// TIA Portal V20 export
// export: Created 2025-12-01T14:57:00.3125225Z, ExportSetting None, DisplayName Totally Integrated Automation Portal, DisplayVersion V20 Update 3, DisplayName TIA Portal Openness, DisplayVersion V20 Update 3, DisplayName TIA Portal Version Control Interface, DisplayVersion V20 Update 3, DisplayName STEP 7 Professional, DisplayVersion V20 Update 3, DisplayName STEP 7 Safety, DisplayVersion V20 Update 2, DisplayName WinCC Basic/Comfort/Advanced, DisplayVersion V20 Update 3, DisplayName WinCC Professional, DisplayVersion V20 Update 3, DisplayName WinCC Unified, DisplayVersion V20 Update 3
FUNCTION "FC450_TL_TR_E1_S2_Pres" : Void   // FC450, LAD
{ S7_Optimized_Access := 'FALSE' }
AUTHOR : TLigero
NAME : 20160512
VERSION : 4.0
// stored: AutoNumber false, SetENOAutomatically false
   VAR_INPUT
      Mesa : UInt;
      En_Tension : Bool;
      PhsMx : Bool;
      Termico_E1 : Bool;
      Termico_S2 : Bool;
      PosTR_E1 : Bool;
      PosTR_S2 : Bool;
      Avance_E1 : Bool;
      Avance_S2 : Bool;
      AVTF_MAnt_Mx : Bool;   // Aviso de transferencia de la mesa anterior
      PTF_Mx_MSig : Bool;   // Permiso de transferencia de la mesa siguiente
      NXT_Avance : Bool;   // Avance de la mesa siguiente
      V_CNT_pHsMx : UDInt;
      V_CNT_ApHsMx : UDInt;
      V_Paro : UDInt;
      V_TOut_Tx_Mx : UDInt;
      V_TOut_transfer : UDInt;
   END_VAR
   VAR_OUTPUT
      PTF_MAnt_Mx : Bool;   // carga ok a la mesa anterior
      AVTF_Mx_MSig : Bool;   // Aviso de transferencia a la mesa siguiente
      NXT_Descarga_Act : Bool;   // descarga activa a la mesa siguiente
   END_VAR
   VAR_TEMP
      Mem_CNT_Tmp_Paro_Tx : Bool;
      Mem_CNT_Pres_entrada : Bool;
      Mem_CNT_Aus_salida : Bool;
      tout_atasco : Bool;
      tout_transfer : Bool;
      TEMP_MA_TR_Pos_E1 : Bool;
      TEMP_MA_TR_Pos_S2 : Bool;
      ok_tension : Bool;
   END_VAR
   VAR_TEMP   // added for the SCL form of the ladder/FBD networks
      _w1 : Bool;
   END_VAR
BEGIN

REGION Network 1: Marca General Error
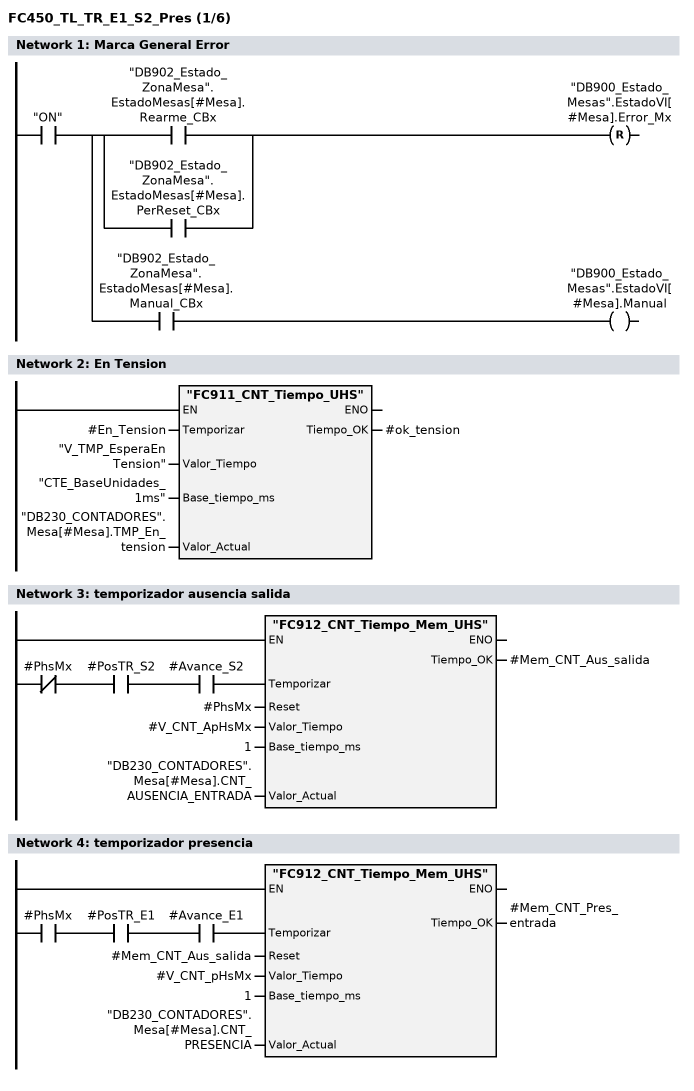
   RUNG wire#powerrail
      Contact( "ON" )
      wire#w1
      Contact( "DB902_Estado_ZonaMesa".EstadoMesas[#Mesa].Rearme_CBx )
      wire#w2
      R_Coil( "DB900_Estado_Mesas".EstadoVI[#Mesa].Error_Mx )
   END_RUNG
   RUNG wire#w1
      Contact( "DB902_Estado_ZonaMesa".EstadoMesas[#Mesa].PerReset_CBx )
   END_RUNG wire#w2
   RUNG wire#w1
      Contact( "DB902_Estado_ZonaMesa".EstadoMesas[#Mesa].Manual_CBx )
      Coil( "DB900_Estado_Mesas".EstadoVI[#Mesa].Manual )
   END_RUNG
   // the same network as SCL:
   IF "ON" AND ("DB902_Estado_ZonaMesa".EstadoMesas[#Mesa].Rearme_CBx OR "DB902_Estado_ZonaMesa".EstadoMesas[#Mesa].PerReset_CBx) THEN
       "DB900_Estado_Mesas".EstadoVI[#Mesa].Error_Mx := FALSE;
   END_IF;
   "DB900_Estado_Mesas".EstadoVI[#Mesa].Manual := "ON" AND "DB902_Estado_ZonaMesa".EstadoMesas[#Mesa].Manual_CBx;
END_REGION

REGION Network 2: En Tension
   RUNG wire#powerrail
      "FC911_CNT_Tiempo_UHS"(Temporizar := #En_Tension, Valor_Tiempo := "V_TMP_EsperaEnTension", Base_tiempo_ms := "CTE_BaseUnidades_1ms", Valor_Actual := "DB230_CONTADORES".Mesa[#Mesa].TMP_En_tension, Tiempo_OK => #ok_tension)
   END_RUNG
   // the same network as SCL:
   "FC911_CNT_Tiempo_UHS"(Temporizar := #En_Tension,
                          Valor_Tiempo := "V_TMP_EsperaEnTension",
                          Base_tiempo_ms := "CTE_BaseUnidades_1ms",
                          Valor_Actual := "DB230_CONTADORES".Mesa[#Mesa].TMP_En_tension,
                          Tiempo_OK => #ok_tension);
END_REGION

REGION Network 3: temporizador ausencia salida
   RUNG wire#powerrail
      "FC912_CNT_Tiempo_Mem_UHS"(Temporizar := wire#w1, Reset := #PhsMx, Valor_Tiempo := #V_CNT_ApHsMx, Base_tiempo_ms := 1, Valor_Actual := "DB230_CONTADORES".Mesa[#Mesa].CNT_AUSENCIA_ENTRADA, Tiempo_OK => #Mem_CNT_Aus_salida)
   END_RUNG
   RUNG wire#powerrail
      I_Contact( #PhsMx )
      Contact( #PosTR_S2 )
      Contact( #Avance_S2 )
   END_RUNG wire#w1
   // the same network as SCL:
   "FC912_CNT_Tiempo_Mem_UHS"(Temporizar := NOT #PhsMx AND #PosTR_S2 AND #Avance_S2,
                           Reset := #PhsMx,
                           Valor_Tiempo := #V_CNT_ApHsMx,
                           Base_tiempo_ms := 1,
                           Valor_Actual := "DB230_CONTADORES".Mesa[#Mesa].CNT_AUSENCIA_ENTRADA,
                           Tiempo_OK => #Mem_CNT_Aus_salida);
END_REGION

REGION Network 4: temporizador presencia
   RUNG wire#powerrail
      "FC912_CNT_Tiempo_Mem_UHS"(Temporizar := wire#w1, Reset := #Mem_CNT_Aus_salida, Valor_Tiempo := #V_CNT_pHsMx, Base_tiempo_ms := 1, Valor_Actual := "DB230_CONTADORES".Mesa[#Mesa].CNT_PRESENCIA, Tiempo_OK => #Mem_CNT_Pres_entrada)
   END_RUNG
   RUNG wire#powerrail
      Contact( #PhsMx )
      Contact( #PosTR_E1 )
      Contact( #Avance_E1 )
   END_RUNG wire#w1
   // the same network as SCL:
   "FC912_CNT_Tiempo_Mem_UHS"(Temporizar := #PhsMx AND #PosTR_E1 AND #Avance_E1,
                           Reset := #Mem_CNT_Aus_salida,
                           Valor_Tiempo := #V_CNT_pHsMx,
                           Base_tiempo_ms := 1,
                           Valor_Actual := "DB230_CONTADORES".Mesa[#Mesa].CNT_PRESENCIA,
                           Tiempo_OK => #Mem_CNT_Pres_entrada);
END_REGION

REGION Network 5: temporizador PARO
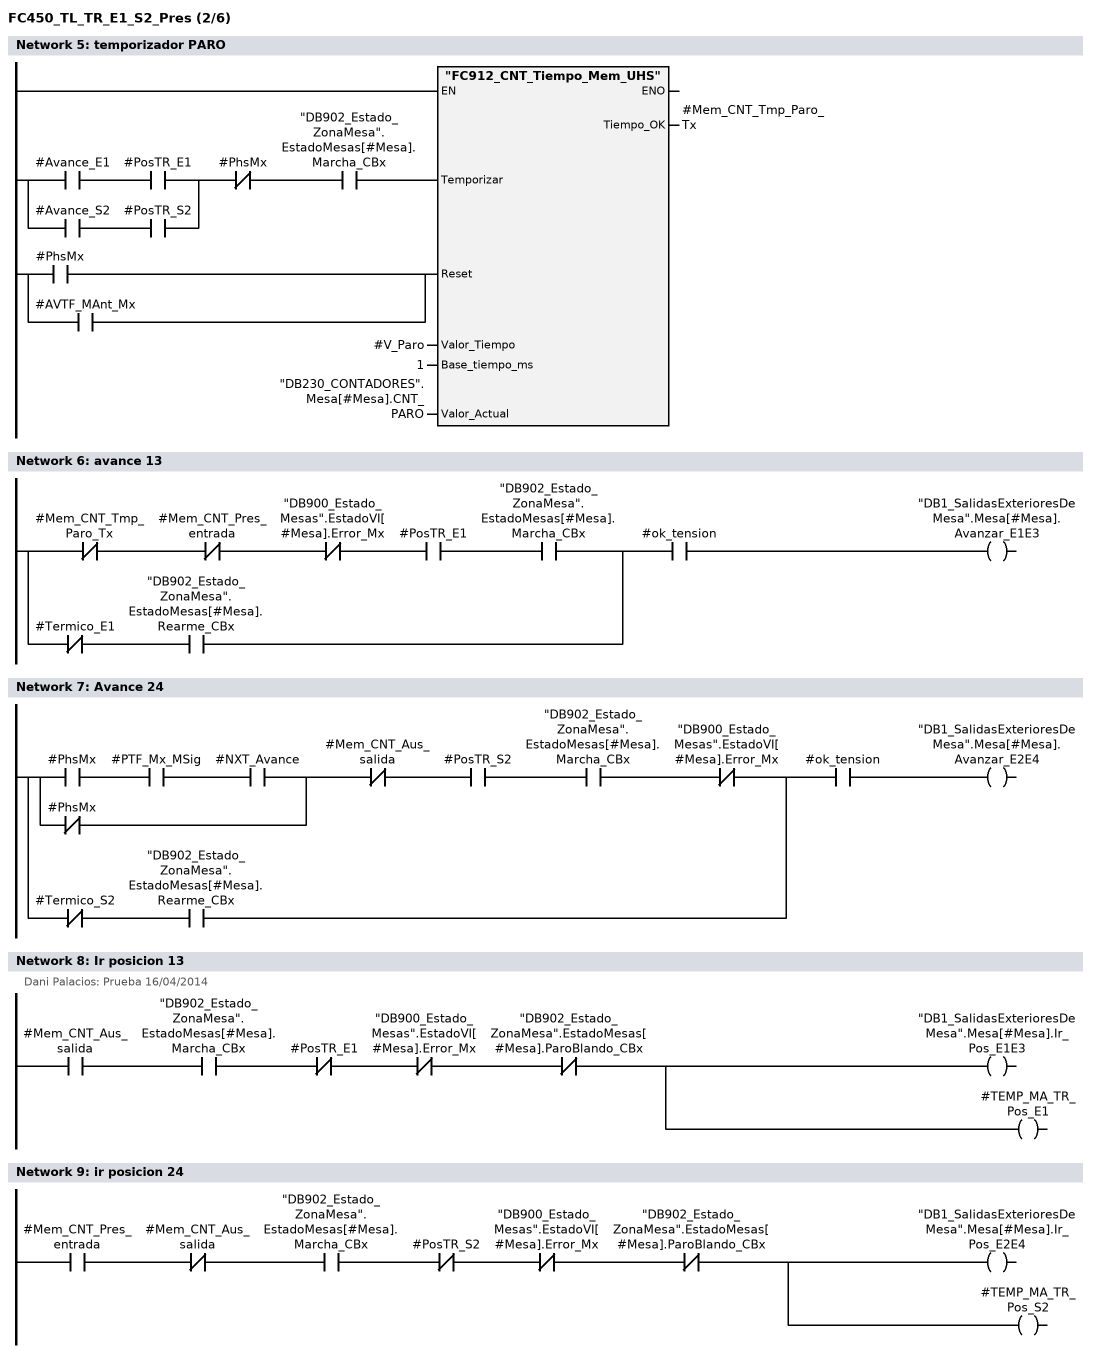
   RUNG wire#powerrail
      "FC912_CNT_Tiempo_Mem_UHS"(Temporizar := wire#w2, Reset := wire#w3, Valor_Tiempo := #V_Paro, Base_tiempo_ms := 1, Valor_Actual := "DB230_CONTADORES".Mesa[#Mesa].CNT_PARO, Tiempo_OK => #Mem_CNT_Tmp_Paro_Tx)
   END_RUNG
   RUNG wire#powerrail
      Contact( #Avance_E1 )
      Contact( #PosTR_E1 )
      wire#w1
      I_Contact( #PhsMx )
      Contact( "DB902_Estado_ZonaMesa".EstadoMesas[#Mesa].Marcha_CBx )
   END_RUNG wire#w2
   RUNG wire#powerrail
      Contact( #Avance_S2 )
      Contact( #PosTR_S2 )
   END_RUNG wire#w1
   RUNG wire#powerrail
      Contact( #PhsMx )
   END_RUNG wire#w3
   RUNG wire#powerrail
      Contact( #AVTF_MAnt_Mx )
   END_RUNG wire#w3
   // the same network as SCL:
   "FC912_CNT_Tiempo_Mem_UHS"(Temporizar := ((#Avance_E1 AND #PosTR_E1) OR (#Avance_S2 AND #PosTR_S2)) AND NOT #PhsMx AND "DB902_Estado_ZonaMesa".EstadoMesas[#Mesa].Marcha_CBx,
                           Reset := #PhsMx OR #AVTF_MAnt_Mx,
                           Valor_Tiempo := #V_Paro,
                           Base_tiempo_ms := 1,
                           Valor_Actual := "DB230_CONTADORES".Mesa[#Mesa].CNT_PARO,
                           Tiempo_OK => #Mem_CNT_Tmp_Paro_Tx);
END_REGION

REGION Network 6: avance 13
   RUNG wire#powerrail
      I_Contact( #Mem_CNT_Tmp_Paro_Tx )
      I_Contact( #Mem_CNT_Pres_entrada )
      I_Contact( "DB900_Estado_Mesas".EstadoVI[#Mesa].Error_Mx )
      Contact( #PosTR_E1 )
      Contact( "DB902_Estado_ZonaMesa".EstadoMesas[#Mesa].Marcha_CBx )
      wire#w1
      Contact( #ok_tension )
      Coil( "DB1_SalidasExterioresDeMesa".Mesa[#Mesa].Avanzar_E1E3 )
   END_RUNG
   RUNG wire#powerrail
      I_Contact( #Termico_E1 )
      Contact( "DB902_Estado_ZonaMesa".EstadoMesas[#Mesa].Rearme_CBx )
   END_RUNG wire#w1
   // the same network as SCL:
   "DB1_SalidasExterioresDeMesa".Mesa[#Mesa].Avanzar_E1E3 := ((NOT #Mem_CNT_Tmp_Paro_Tx AND NOT #Mem_CNT_Pres_entrada AND NOT "DB900_Estado_Mesas".EstadoVI[#Mesa].Error_Mx AND #PosTR_E1 AND "DB902_Estado_ZonaMesa".EstadoMesas[#Mesa].Marcha_CBx) OR (NOT #Termico_E1 AND "DB902_Estado_ZonaMesa".EstadoMesas[#Mesa].Rearme_CBx)) AND #ok_tension;
END_REGION

REGION Network 7: Avance 24
   RUNG wire#powerrail
      Contact( #PhsMx )
      Contact( #PTF_Mx_MSig )
      Contact( #NXT_Avance )
      wire#w1
      I_Contact( #Mem_CNT_Aus_salida )
      Contact( #PosTR_S2 )
      Contact( "DB902_Estado_ZonaMesa".EstadoMesas[#Mesa].Marcha_CBx )
      I_Contact( "DB900_Estado_Mesas".EstadoVI[#Mesa].Error_Mx )
      wire#w2
      Contact( #ok_tension )
      Coil( "DB1_SalidasExterioresDeMesa".Mesa[#Mesa].Avanzar_E2E4 )
   END_RUNG
   RUNG wire#powerrail
      I_Contact( #PhsMx )
   END_RUNG wire#w1
   RUNG wire#powerrail
      I_Contact( #Termico_S2 )
      Contact( "DB902_Estado_ZonaMesa".EstadoMesas[#Mesa].Rearme_CBx )
   END_RUNG wire#w2
   // the same network as SCL:
   "DB1_SalidasExterioresDeMesa".Mesa[#Mesa].Avanzar_E2E4 := ((((#PhsMx AND #PTF_Mx_MSig AND #NXT_Avance) OR NOT #PhsMx) AND NOT #Mem_CNT_Aus_salida AND #PosTR_S2 AND "DB902_Estado_ZonaMesa".EstadoMesas[#Mesa].Marcha_CBx AND NOT "DB900_Estado_Mesas".EstadoVI[#Mesa].Error_Mx) OR (NOT #Termico_S2 AND "DB902_Estado_ZonaMesa".EstadoMesas[#Mesa].Rearme_CBx)) AND #ok_tension;
END_REGION

REGION Network 8: Ir posicion 13
   // Dani Palacios: Prueba 16/04/2014
   RUNG wire#powerrail
      Contact( #Mem_CNT_Aus_salida )
      Contact( "DB902_Estado_ZonaMesa".EstadoMesas[#Mesa].Marcha_CBx )
      I_Contact( #PosTR_E1 )
      I_Contact( "DB900_Estado_Mesas".EstadoVI[#Mesa].Error_Mx )
      I_Contact( "DB902_Estado_ZonaMesa".EstadoMesas[#Mesa].ParoBlando_CBx )
      wire#w1
      Coil( "DB1_SalidasExterioresDeMesa".Mesa[#Mesa].Ir_Pos_E1E3 )
   END_RUNG
   RUNG wire#w1
      Coil( #TEMP_MA_TR_Pos_E1 )
   END_RUNG
   // the same network as SCL:
   #_w1 := #Mem_CNT_Aus_salida AND "DB902_Estado_ZonaMesa".EstadoMesas[#Mesa].Marcha_CBx AND NOT #PosTR_E1 AND NOT "DB900_Estado_Mesas".EstadoVI[#Mesa].Error_Mx AND NOT "DB902_Estado_ZonaMesa".EstadoMesas[#Mesa].ParoBlando_CBx;
   "DB1_SalidasExterioresDeMesa".Mesa[#Mesa].Ir_Pos_E1E3 := #Mem_CNT_Aus_salida AND "DB902_Estado_ZonaMesa".EstadoMesas[#Mesa].Marcha_CBx AND NOT #PosTR_E1 AND NOT "DB900_Estado_Mesas".EstadoVI[#Mesa].Error_Mx AND NOT "DB902_Estado_ZonaMesa".EstadoMesas[#Mesa].ParoBlando_CBx;
   #TEMP_MA_TR_Pos_E1 := #_w1;
END_REGION

REGION Network 9: ir posicion 24
   RUNG wire#powerrail
      Contact( #Mem_CNT_Pres_entrada )
      I_Contact( #Mem_CNT_Aus_salida )
      Contact( "DB902_Estado_ZonaMesa".EstadoMesas[#Mesa].Marcha_CBx )
      I_Contact( #PosTR_S2 )
      I_Contact( "DB900_Estado_Mesas".EstadoVI[#Mesa].Error_Mx )
      I_Contact( "DB902_Estado_ZonaMesa".EstadoMesas[#Mesa].ParoBlando_CBx )
      wire#w1
      Coil( "DB1_SalidasExterioresDeMesa".Mesa[#Mesa].Ir_Pos_E2E4 )
   END_RUNG
   RUNG wire#w1
      Coil( #TEMP_MA_TR_Pos_S2 )
   END_RUNG
   // the same network as SCL:
   #_w1 := #Mem_CNT_Pres_entrada AND NOT #Mem_CNT_Aus_salida AND "DB902_Estado_ZonaMesa".EstadoMesas[#Mesa].Marcha_CBx AND NOT #PosTR_S2 AND NOT "DB900_Estado_Mesas".EstadoVI[#Mesa].Error_Mx AND NOT "DB902_Estado_ZonaMesa".EstadoMesas[#Mesa].ParoBlando_CBx;
   "DB1_SalidasExterioresDeMesa".Mesa[#Mesa].Ir_Pos_E2E4 := #Mem_CNT_Pres_entrada AND NOT #Mem_CNT_Aus_salida AND "DB902_Estado_ZonaMesa".EstadoMesas[#Mesa].Marcha_CBx AND NOT #PosTR_S2 AND NOT "DB900_Estado_Mesas".EstadoVI[#Mesa].Error_Mx AND NOT "DB902_Estado_ZonaMesa".EstadoMesas[#Mesa].ParoBlando_CBx;
   #TEMP_MA_TR_Pos_S2 := #_w1;
END_REGION

REGION Network 10: nxt avtf
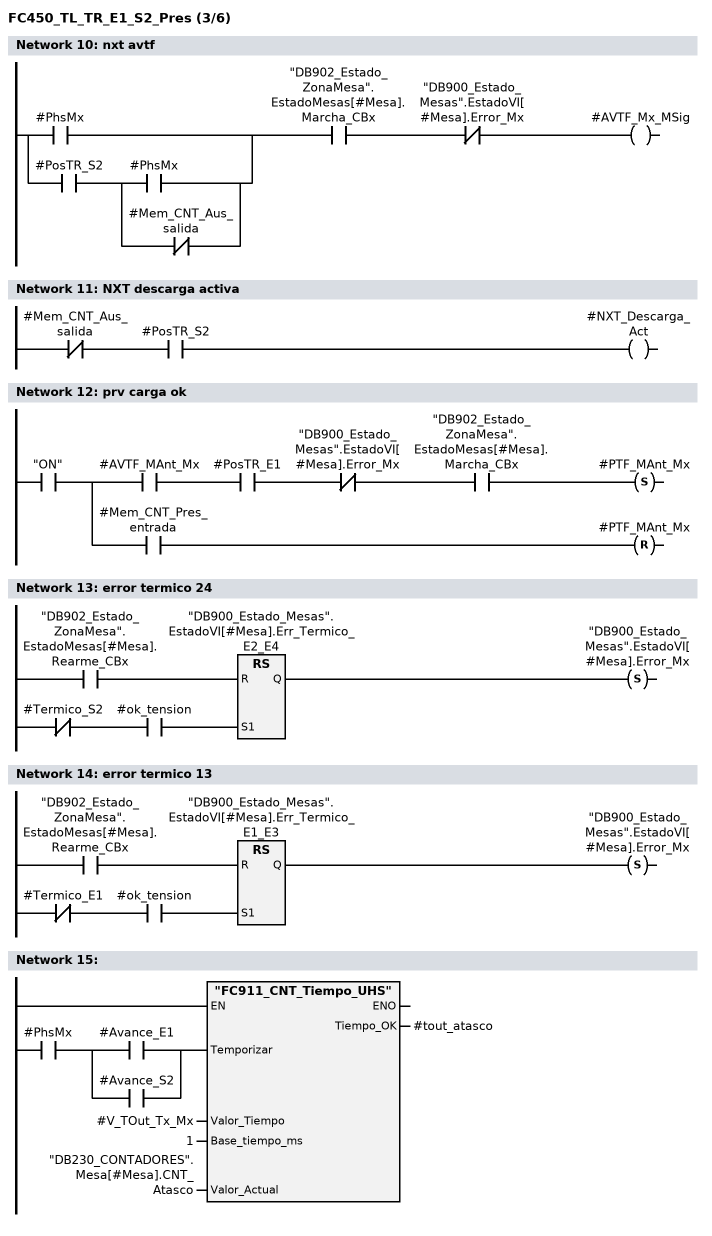
   RUNG wire#powerrail
      Contact( #PhsMx )
      wire#w1
      Contact( "DB902_Estado_ZonaMesa".EstadoMesas[#Mesa].Marcha_CBx )
      I_Contact( "DB900_Estado_Mesas".EstadoVI[#Mesa].Error_Mx )
      Coil( #AVTF_Mx_MSig )
   END_RUNG
   RUNG wire#powerrail
      Contact( #PosTR_S2 )
      wire#w2
      Contact( #PhsMx )
   END_RUNG wire#w1
   RUNG wire#w2
      I_Contact( #Mem_CNT_Aus_salida )
   END_RUNG wire#w1
   // the same network as SCL:
   #AVTF_Mx_MSig := (#PhsMx OR (#PosTR_S2 AND (#PhsMx OR NOT #Mem_CNT_Aus_salida))) AND "DB902_Estado_ZonaMesa".EstadoMesas[#Mesa].Marcha_CBx AND NOT "DB900_Estado_Mesas".EstadoVI[#Mesa].Error_Mx;
END_REGION

REGION Network 11: NXT descarga activa
   RUNG wire#powerrail
      I_Contact( #Mem_CNT_Aus_salida )
      Contact( #PosTR_S2 )
      Coil( #NXT_Descarga_Act )
   END_RUNG
   // the same network as SCL:
   #NXT_Descarga_Act := NOT #Mem_CNT_Aus_salida AND #PosTR_S2;
END_REGION

REGION Network 12: prv carga ok
   RUNG wire#powerrail
      Contact( "ON" )
      wire#w1
      Contact( #AVTF_MAnt_Mx )
      Contact( #PosTR_E1 )
      I_Contact( "DB900_Estado_Mesas".EstadoVI[#Mesa].Error_Mx )
      Contact( "DB902_Estado_ZonaMesa".EstadoMesas[#Mesa].Marcha_CBx )
      S_Coil( #PTF_MAnt_Mx )
   END_RUNG
   RUNG wire#w1
      Contact( #Mem_CNT_Pres_entrada )
      R_Coil( #PTF_MAnt_Mx )
   END_RUNG
   // the same network as SCL:
   IF "ON" AND #AVTF_MAnt_Mx AND #PosTR_E1 AND NOT "DB900_Estado_Mesas".EstadoVI[#Mesa].Error_Mx AND "DB902_Estado_ZonaMesa".EstadoMesas[#Mesa].Marcha_CBx THEN
       #PTF_MAnt_Mx := TRUE;
   END_IF;
   IF "ON" AND #Mem_CNT_Pres_entrada THEN #PTF_MAnt_Mx := FALSE; END_IF;
END_REGION

REGION Network 13: error termico 24
   RUNG wire#powerrail
      Contact( "DB902_Estado_ZonaMesa".EstadoMesas[#Mesa].Rearme_CBx )
      S_RS(operand := "DB900_Estado_Mesas".EstadoVI[#Mesa].Err_Termico_E2_E4, s1 := wire#w1)
      S_Coil( "DB900_Estado_Mesas".EstadoVI[#Mesa].Error_Mx )
   END_RUNG
   RUNG wire#powerrail
      I_Contact( #Termico_S2 )
      Contact( #ok_tension )
   END_RUNG wire#w1
   // the same network as SCL:
   IF "DB902_Estado_ZonaMesa".EstadoMesas[#Mesa].Rearme_CBx THEN
       "DB900_Estado_Mesas".EstadoVI[#Mesa].Err_Termico_E2_E4 := FALSE;   // RS flip-flop
   END_IF;
   IF NOT #Termico_S2 AND #ok_tension THEN
       "DB900_Estado_Mesas".EstadoVI[#Mesa].Err_Termico_E2_E4 := TRUE;
   END_IF;
   IF "DB900_Estado_Mesas".EstadoVI[#Mesa].Err_Termico_E2_E4 THEN
       "DB900_Estado_Mesas".EstadoVI[#Mesa].Error_Mx := TRUE;
   END_IF;
END_REGION

REGION Network 14: error termico 13
   RUNG wire#powerrail
      Contact( "DB902_Estado_ZonaMesa".EstadoMesas[#Mesa].Rearme_CBx )
      S_RS(operand := "DB900_Estado_Mesas".EstadoVI[#Mesa].Err_Termico_E1_E3, s1 := wire#w1)
      S_Coil( "DB900_Estado_Mesas".EstadoVI[#Mesa].Error_Mx )
   END_RUNG
   RUNG wire#powerrail
      I_Contact( #Termico_E1 )
      Contact( #ok_tension )
   END_RUNG wire#w1
   // the same network as SCL:
   IF "DB902_Estado_ZonaMesa".EstadoMesas[#Mesa].Rearme_CBx THEN
       "DB900_Estado_Mesas".EstadoVI[#Mesa].Err_Termico_E1_E3 := FALSE;   // RS flip-flop
   END_IF;
   IF NOT #Termico_E1 AND #ok_tension THEN
       "DB900_Estado_Mesas".EstadoVI[#Mesa].Err_Termico_E1_E3 := TRUE;
   END_IF;
   IF "DB900_Estado_Mesas".EstadoVI[#Mesa].Err_Termico_E1_E3 THEN
       "DB900_Estado_Mesas".EstadoVI[#Mesa].Error_Mx := TRUE;
   END_IF;
END_REGION

REGION Network 15
   RUNG wire#powerrail
      "FC911_CNT_Tiempo_UHS"(Temporizar := wire#w2, Valor_Tiempo := #V_TOut_Tx_Mx, Base_tiempo_ms := 1, Valor_Actual := "DB230_CONTADORES".Mesa[#Mesa].CNT_Atasco, Tiempo_OK => #tout_atasco)
   END_RUNG
   RUNG wire#powerrail
      Contact( #PhsMx )
      wire#w1
      Contact( #Avance_E1 )
   END_RUNG wire#w2
   RUNG wire#w1
      Contact( #Avance_S2 )
   END_RUNG wire#w2
   // the same network as SCL:
   "FC911_CNT_Tiempo_UHS"(Temporizar := #PhsMx AND (#Avance_E1 OR #Avance_S2),
                          Valor_Tiempo := #V_TOut_Tx_Mx,
                          Base_tiempo_ms := 1,
                          Valor_Actual := "DB230_CONTADORES".Mesa[#Mesa].CNT_Atasco,
                          Tiempo_OK => #tout_atasco);
END_REGION

REGION Network 16: Marca General Error
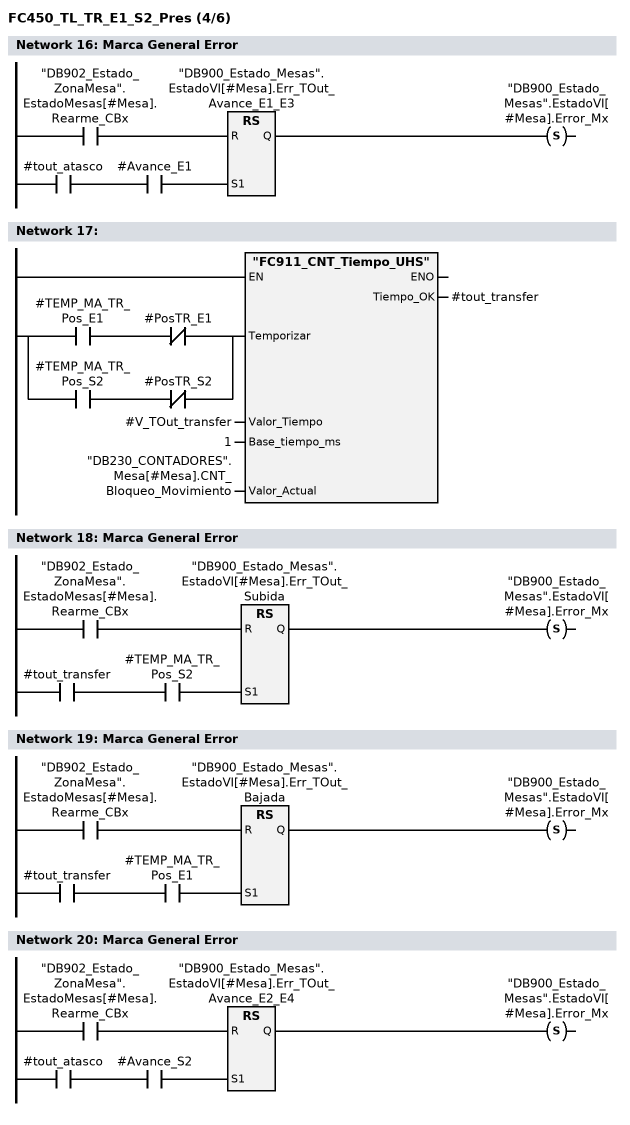
   RUNG wire#powerrail
      Contact( "DB902_Estado_ZonaMesa".EstadoMesas[#Mesa].Rearme_CBx )
      S_RS(operand := "DB900_Estado_Mesas".EstadoVI[#Mesa].Err_TOut_Avance_E1_E3, s1 := wire#w1)
      S_Coil( "DB900_Estado_Mesas".EstadoVI[#Mesa].Error_Mx )
   END_RUNG
   RUNG wire#powerrail
      Contact( #tout_atasco )
      Contact( #Avance_E1 )
   END_RUNG wire#w1
   // the same network as SCL:
   IF "DB902_Estado_ZonaMesa".EstadoMesas[#Mesa].Rearme_CBx THEN
       "DB900_Estado_Mesas".EstadoVI[#Mesa].Err_TOut_Avance_E1_E3 := FALSE;   // RS flip-flop
   END_IF;
   IF #tout_atasco AND #Avance_E1 THEN
       "DB900_Estado_Mesas".EstadoVI[#Mesa].Err_TOut_Avance_E1_E3 := TRUE;
   END_IF;
   IF "DB900_Estado_Mesas".EstadoVI[#Mesa].Err_TOut_Avance_E1_E3 THEN
       "DB900_Estado_Mesas".EstadoVI[#Mesa].Error_Mx := TRUE;
   END_IF;
END_REGION

REGION Network 17
   RUNG wire#powerrail
      "FC911_CNT_Tiempo_UHS"(Temporizar := wire#w1, Valor_Tiempo := #V_TOut_transfer, Base_tiempo_ms := 1, Valor_Actual := "DB230_CONTADORES".Mesa[#Mesa].CNT_Bloqueo_Movimiento, Tiempo_OK => #tout_transfer)
   END_RUNG
   RUNG wire#powerrail
      Contact( #TEMP_MA_TR_Pos_E1 )
      I_Contact( #PosTR_E1 )
   END_RUNG wire#w1
   RUNG wire#powerrail
      Contact( #TEMP_MA_TR_Pos_S2 )
      I_Contact( #PosTR_S2 )
   END_RUNG wire#w1
   // the same network as SCL:
   "FC911_CNT_Tiempo_UHS"(Temporizar := (#TEMP_MA_TR_Pos_E1 AND NOT #PosTR_E1) OR (#TEMP_MA_TR_Pos_S2 AND NOT #PosTR_S2),
                          Valor_Tiempo := #V_TOut_transfer,
                          Base_tiempo_ms := 1,
                          Valor_Actual := "DB230_CONTADORES".Mesa[#Mesa].CNT_Bloqueo_Movimiento,
                          Tiempo_OK => #tout_transfer);
END_REGION

REGION Network 18: Marca General Error
   RUNG wire#powerrail
      Contact( "DB902_Estado_ZonaMesa".EstadoMesas[#Mesa].Rearme_CBx )
      S_RS(operand := "DB900_Estado_Mesas".EstadoVI[#Mesa].Err_TOut_Subida, s1 := wire#w1)
      S_Coil( "DB900_Estado_Mesas".EstadoVI[#Mesa].Error_Mx )
   END_RUNG
   RUNG wire#powerrail
      Contact( #tout_transfer )
      Contact( #TEMP_MA_TR_Pos_S2 )
   END_RUNG wire#w1
   // the same network as SCL:
   IF "DB902_Estado_ZonaMesa".EstadoMesas[#Mesa].Rearme_CBx THEN
       "DB900_Estado_Mesas".EstadoVI[#Mesa].Err_TOut_Subida := FALSE;   // RS flip-flop
   END_IF;
   IF #tout_transfer AND #TEMP_MA_TR_Pos_S2 THEN
       "DB900_Estado_Mesas".EstadoVI[#Mesa].Err_TOut_Subida := TRUE;
   END_IF;
   IF "DB900_Estado_Mesas".EstadoVI[#Mesa].Err_TOut_Subida THEN
       "DB900_Estado_Mesas".EstadoVI[#Mesa].Error_Mx := TRUE;
   END_IF;
END_REGION

REGION Network 19: Marca General Error
   RUNG wire#powerrail
      Contact( "DB902_Estado_ZonaMesa".EstadoMesas[#Mesa].Rearme_CBx )
      S_RS(operand := "DB900_Estado_Mesas".EstadoVI[#Mesa].Err_TOut_Bajada, s1 := wire#w1)
      S_Coil( "DB900_Estado_Mesas".EstadoVI[#Mesa].Error_Mx )
   END_RUNG
   RUNG wire#powerrail
      Contact( #tout_transfer )
      Contact( #TEMP_MA_TR_Pos_E1 )
   END_RUNG wire#w1
   // the same network as SCL:
   IF "DB902_Estado_ZonaMesa".EstadoMesas[#Mesa].Rearme_CBx THEN
       "DB900_Estado_Mesas".EstadoVI[#Mesa].Err_TOut_Bajada := FALSE;   // RS flip-flop
   END_IF;
   IF #tout_transfer AND #TEMP_MA_TR_Pos_E1 THEN
       "DB900_Estado_Mesas".EstadoVI[#Mesa].Err_TOut_Bajada := TRUE;
   END_IF;
   IF "DB900_Estado_Mesas".EstadoVI[#Mesa].Err_TOut_Bajada THEN
       "DB900_Estado_Mesas".EstadoVI[#Mesa].Error_Mx := TRUE;
   END_IF;
END_REGION

REGION Network 20: Marca General Error
   RUNG wire#powerrail
      Contact( "DB902_Estado_ZonaMesa".EstadoMesas[#Mesa].Rearme_CBx )
      S_RS(operand := "DB900_Estado_Mesas".EstadoVI[#Mesa].Err_TOut_Avance_E2_E4, s1 := wire#w1)
      S_Coil( "DB900_Estado_Mesas".EstadoVI[#Mesa].Error_Mx )
   END_RUNG
   RUNG wire#powerrail
      Contact( #tout_atasco )
      Contact( #Avance_S2 )
   END_RUNG wire#w1
   // the same network as SCL:
   IF "DB902_Estado_ZonaMesa".EstadoMesas[#Mesa].Rearme_CBx THEN
       "DB900_Estado_Mesas".EstadoVI[#Mesa].Err_TOut_Avance_E2_E4 := FALSE;   // RS flip-flop
   END_IF;
   IF #tout_atasco AND #Avance_S2 THEN
       "DB900_Estado_Mesas".EstadoVI[#Mesa].Err_TOut_Avance_E2_E4 := TRUE;
   END_IF;
   IF "DB900_Estado_Mesas".EstadoVI[#Mesa].Err_TOut_Avance_E2_E4 THEN
       "DB900_Estado_Mesas".EstadoVI[#Mesa].Error_Mx := TRUE;
   END_IF;
END_REGION

REGION Network 21: Entradas Mesas
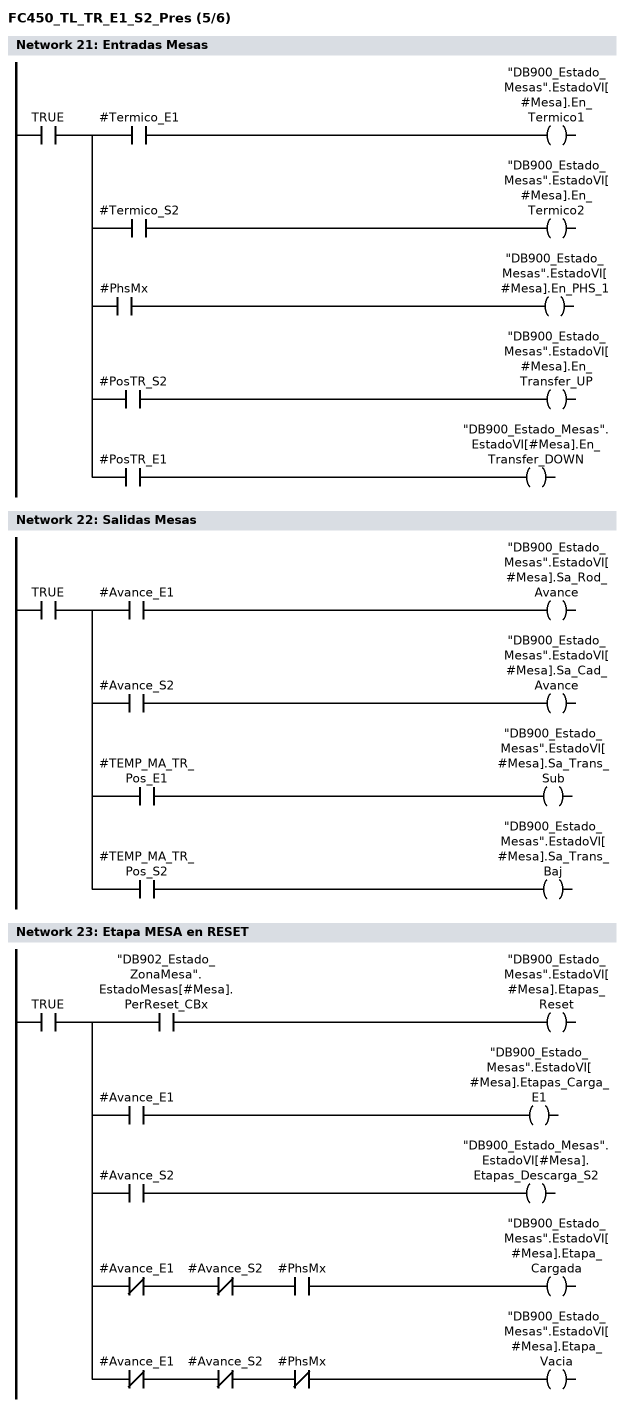
   RUNG wire#powerrail
      Contact( TRUE )
      wire#w1
      Contact( #Termico_E1 )
      Coil( "DB900_Estado_Mesas".EstadoVI[#Mesa].En_Termico1 )
   END_RUNG
   RUNG wire#w1
      Contact( #Termico_S2 )
      Coil( "DB900_Estado_Mesas".EstadoVI[#Mesa].En_Termico2 )
   END_RUNG
   RUNG wire#w1
      Contact( #PhsMx )
      Coil( "DB900_Estado_Mesas".EstadoVI[#Mesa].En_PHS_1 )
   END_RUNG
   RUNG wire#w1
      Contact( #PosTR_S2 )
      Coil( "DB900_Estado_Mesas".EstadoVI[#Mesa].En_Transfer_UP )
   END_RUNG
   RUNG wire#w1
      Contact( #PosTR_E1 )
      Coil( "DB900_Estado_Mesas".EstadoVI[#Mesa].En_Transfer_DOWN )
   END_RUNG
   // the same network as SCL:
   "DB900_Estado_Mesas".EstadoVI[#Mesa].En_Termico1 := TRUE AND #Termico_E1;
   "DB900_Estado_Mesas".EstadoVI[#Mesa].En_Termico2 := TRUE AND #Termico_S2;
   "DB900_Estado_Mesas".EstadoVI[#Mesa].En_PHS_1 := TRUE AND #PhsMx;
   "DB900_Estado_Mesas".EstadoVI[#Mesa].En_Transfer_UP := TRUE AND #PosTR_S2;
   "DB900_Estado_Mesas".EstadoVI[#Mesa].En_Transfer_DOWN := TRUE AND #PosTR_E1;
END_REGION

REGION Network 22: Salidas Mesas
   RUNG wire#powerrail
      Contact( TRUE )
      wire#w1
      Contact( #Avance_E1 )
      Coil( "DB900_Estado_Mesas".EstadoVI[#Mesa].Sa_Rod_Avance )
   END_RUNG
   RUNG wire#w1
      Contact( #Avance_S2 )
      Coil( "DB900_Estado_Mesas".EstadoVI[#Mesa].Sa_Cad_Avance )
   END_RUNG
   RUNG wire#w1
      Contact( #TEMP_MA_TR_Pos_E1 )
      Coil( "DB900_Estado_Mesas".EstadoVI[#Mesa].Sa_Trans_Sub )
   END_RUNG
   RUNG wire#w1
      Contact( #TEMP_MA_TR_Pos_S2 )
      Coil( "DB900_Estado_Mesas".EstadoVI[#Mesa].Sa_Trans_Baj )
   END_RUNG
   // the same network as SCL:
   "DB900_Estado_Mesas".EstadoVI[#Mesa].Sa_Rod_Avance := TRUE AND #Avance_E1;
   "DB900_Estado_Mesas".EstadoVI[#Mesa].Sa_Cad_Avance := TRUE AND #Avance_S2;
   "DB900_Estado_Mesas".EstadoVI[#Mesa].Sa_Trans_Sub := TRUE AND #TEMP_MA_TR_Pos_E1;
   "DB900_Estado_Mesas".EstadoVI[#Mesa].Sa_Trans_Baj := TRUE AND #TEMP_MA_TR_Pos_S2;
END_REGION

REGION Network 23: Etapa MESA en RESET
   RUNG wire#powerrail
      Contact( TRUE )
      wire#w1
      Contact( "DB902_Estado_ZonaMesa".EstadoMesas[#Mesa].PerReset_CBx )
      Coil( "DB900_Estado_Mesas".EstadoVI[#Mesa].Etapas_Reset )
   END_RUNG
   RUNG wire#w1
      Contact( #Avance_E1 )
      Coil( "DB900_Estado_Mesas".EstadoVI[#Mesa].Etapas_Carga_E1 )
   END_RUNG
   RUNG wire#w1
      Contact( #Avance_S2 )
      Coil( "DB900_Estado_Mesas".EstadoVI[#Mesa].Etapas_Descarga_S2 )
   END_RUNG
   RUNG wire#w1
      I_Contact( #Avance_E1 )
      I_Contact( #Avance_S2 )
      Contact( #PhsMx )
      Coil( "DB900_Estado_Mesas".EstadoVI[#Mesa].Etapa_Cargada )
   END_RUNG
   RUNG wire#w1
      I_Contact( #Avance_E1 )
      I_Contact( #Avance_S2 )
      I_Contact( #PhsMx )
      Coil( "DB900_Estado_Mesas".EstadoVI[#Mesa].Etapa_Vacia )
   END_RUNG
   // the same network as SCL:
   "DB900_Estado_Mesas".EstadoVI[#Mesa].Etapas_Reset := TRUE AND "DB902_Estado_ZonaMesa".EstadoMesas[#Mesa].PerReset_CBx;
   "DB900_Estado_Mesas".EstadoVI[#Mesa].Etapas_Carga_E1 := TRUE AND #Avance_E1;
   "DB900_Estado_Mesas".EstadoVI[#Mesa].Etapas_Descarga_S2 := TRUE AND #Avance_S2;
   "DB900_Estado_Mesas".EstadoVI[#Mesa].Etapa_Cargada := TRUE AND NOT #Avance_E1 AND NOT #Avance_S2 AND #PhsMx;
   "DB900_Estado_Mesas".EstadoVI[#Mesa].Etapa_Vacia := TRUE AND NOT #Avance_E1 AND NOT #Avance_S2 AND NOT #PhsMx;
END_REGION

REGION Network 24
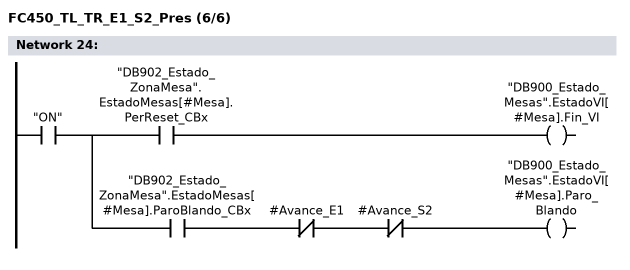
   RUNG wire#powerrail
      Contact( "ON" )
      wire#w1
      Contact( "DB902_Estado_ZonaMesa".EstadoMesas[#Mesa].PerReset_CBx )
      Coil( "DB900_Estado_Mesas".EstadoVI[#Mesa].Fin_VI )
   END_RUNG
   RUNG wire#w1
      Contact( "DB902_Estado_ZonaMesa".EstadoMesas[#Mesa].ParoBlando_CBx )
      I_Contact( #Avance_E1 )
      I_Contact( #Avance_S2 )
      Coil( "DB900_Estado_Mesas".EstadoVI[#Mesa].Paro_Blando )
   END_RUNG
   // the same network as SCL:
   "DB900_Estado_Mesas".EstadoVI[#Mesa].Fin_VI := "ON" AND "DB902_Estado_ZonaMesa".EstadoMesas[#Mesa].PerReset_CBx;
   "DB900_Estado_Mesas".EstadoVI[#Mesa].Paro_Blando := "ON" AND "DB902_Estado_ZonaMesa".EstadoMesas[#Mesa].ParoBlando_CBx AND NOT #Avance_E1 AND NOT #Avance_S2;
END_REGION
END_FUNCTION
